INTERFACE ITF_LiftActuator

METHOD ExtendActuator : BOOL
VAR_INPUT
END_VAR
END_METHOD

METHOD RetractActuator : BOOL
VAR_INPUT
END_VAR
END_METHOD

END_INTERFACE

(* stored: Version 1.1.0.1
   Itf ITF_LiftActuator: Id {bf46c465-a154-4fb4-8abd-ed2c37f02185}
   Method ExtendActuator: Id {73a03185-251c-4d08-b80c-94b096a85c38}
   Method RetractActuator: Id {8c472bbf-adb5-4db8-8471-4d8a593a300e} *)
